(* CODESYS project IDE.xml
   cds-sync-save-after-import: True
   cds-sync-backup-name: cds-text-sync-reference-project
   cds-sync-enable-logging: True
   cds-text-sync-multipleApps: True
   cds-sync-backup-binary: True
   cds-sync-export-xml: True
   cds-sync-xml-first: True
   cds-sync-version: 1.7.5
   cds-sync-backup-retention-count: 3
   cds-sync-save-after-export: True
   cds-sync-safety-backup: True
   cds-sync-folder: C:\Workspace\Active\cds-text-sync-reference-project
   cds-sync-silent-mode: False
   cds-sync-pc: LOQ
   cds-daemon-config: {"poll_ms": 10, "deny": ["reset_plc", "reset_plc --kind origin", "create_boot_app", "plc_upload", "source_download"]}
   cds-sync-type-profile: codesys_sp20_plus

Project tree, tasks and I/O mapping:
  PLC : CODESYS Control Win V3 x64, CODESYS, version 3.5.20.10
    application ST_Application
      libraries: Standard, 3.5.22.0 (System); CAA CiA 405, 4.3.0.0 (CODESYS)
      task Task (cyclic, interval t#20ms, priority 1) calls ST_PROGRAMM, ST_PROGRAMM_AUX
      task Profinet_IOTask (cyclic, interval t#1ms, priority 1) calls nothing
      task Profinet_CommunicationTask (cyclic, interval t#10ms, priority 14) calls PN_Controller.CommCycle
      task EtherCAT_Task (cyclic, interval t#4ms, priority 1) calls nothing
      03_Object_POU_ST/
        01_PROGRAMM/
          program ST_PROGRAMM [ST]: ST_METHOD, ST_PROPERTY, ST_ACTION
          program ST_PROGRAMM_AUX [ST]
        02_FunctioanalBlock/
          function block ST_FB [ST]: ST_FB_Action, ST_FB_Method, ST_FB_Property
          function block ST_BLOCK_WITH_INTERFACE [ST]
        03_Function/
          function ST_Function [ST]
          function Empty_impementation_fn [ST]
          function fnBEETWEEN [ST]
        04_Interface/
          interface ITF_Base
          interface ITF_Child: Get_Value
      02_Object_GVL/
        declarations _02_TaskLocalGVL
        global variables _01_GVL
        global variables _03_NVL_sender
      01_Object_DUT/
        data type _04_DUT_UNION
        data type _02_DUT_Enumeration
        data type _03_DUT_Alias
        data type _01_DUT_STRUCTURE
        data type _01_DUT_STRUCTURE2
      04_additional/
        text list TextList
      Symbols
    application LD_Application
      libraries: Standard, 3.5.22.0 (System)
      task Task (cyclic, interval t#20ms, priority 1) calls LD_PROGRAMM, LD2_PROGRAMM
      03_Object_POU_LD/
        01_PROGRAMM/
          program LD_PROGRAMM [LD]
          program LD2_PROGRAMM [?]
        02_FunctionalBlock/
          function block LD_FB [LD]
        03_Function/
          function LD_Function [LD]
    application CFC_Application
      task Task (cyclic, interval t#20ms, priority 1) calls CFC_PROGRAMM, CFC_Page_PROGRAMM
      03_Object_POU_CFC/
        01_PROGRAMM/
          program CFC_PROGRAMM [CFC]
          program CFC_Page_PROGRAMM [CFC]
        02_FunctionalBlock/
          function block CFC_FB [CFC]
        03_Function/
          function CFC_R_TRIG [CFC]
      04_Persistent_vars/
      01_Object_DUT/
        data type _04_DUT_UNION
        data type _02_DUT_Enumeration
        data type _03_DUT_Alias
        data type _01_DUT_STRUCTURE
        data type _01_DUT_STRUCTURE2
    application FBD_Application
      libraries: Standard, 3.5.22.0 (System)
      task Task (cyclic, interval t#20ms, priority 1) calls nothing
      03_Object_POU_FBD/
        01_PROGRAMM/
        02_FunctionalBlock/
          function block FBD_FunctionBlock [FBD]: ST_Method_under_XML
        03_Function/
    Ethernet_Modbus : Ethernet, CODESYS, version 4.2.0.0
      Modbus_TCP_Client : Modbus TCP Client, CODESYS, version 4.5.0.0
        Modbus_TCP_Server : Modbus TCP Server, CODESYS, version 4.5.0.0
            settings: Unit-ID = 255; Channel 0.Function Code = 3; Channel 0.Read Offset = 16#0000; Channel 0.Read Length = 10; Channel 0.Write Offset = 0; Channel 0.Write Length = 0; Channel 0.Cycle Time = 100; Channel 1.Function Code = 16; Channel 1.Read Offset = 0; Channel 1.Read Length = 0; Channel 1.Write Offset = 16#0000; Channel 1.Write Length = 10; Channel 1.Cycle Time = 100
            unmapped channels: Channel 0, Channel 1
    Ethernet_Profinet : Ethernet, CODESYS, version 4.2.0.0
      PN_Controller : PN-Controller, CODESYS, order no. 1, version 4.7.1.0
          settings: First IP Address = [192, 168, 0, 2]; Last IP Address = [192, 168, 0, 254]; Default Subnet Mask = [255, 255, 255, 0]; Default Gateway Address = [0, 0, 0, 0]
        EL6631_0010_V2_0 : EL6631-0010 V2.0, Beckhoff, order no. EL6631-0010, version SW=V1.00, HW=V1.00
            settings: Slave parameters.Identification.IP address = [192,168,0,2]; Slave parameters.Identification.Subnet mask = [255,255,255,0]; Slave parameters.Identification.Default gateway = [0,0,0,0]; Slave parameters.Identification.MAC address = [16#00,16#00,16#00,16#00,16#00,16#00]; Slave parameters.Reduction ratio = 4; Slave parameters.Watchdog interval = 3
            unmapped channels: Inputs PS
    EtherCAT_Master : EtherCAT Master, CODESYS, version 4.10.0.0
      Unidrive_SP_Closed_Loop : Unidrive SP Closed Loop SoftMotion, Control Techniques, version 4.19.0.0
          settings: DC sync0 cycletime = 4000
          unmapped channels: Target Position, Control word, Modes of operation, Actual position, Status word, Modes of operation display
        SM_Drive_EtherCAT_ControlTechniques : SM_Drive_EtherCAT_ControlTechniques, CODESYS, order no. 0, version 4.19.0.0
            settings: wDriveID = 0; fSWMaxVelocity = 60; AddressOffset_8010 = 24; BitOffset_8010 = 0; BitLength_8010 = 16; Address_8010 = '%QW12'; Type_8010 = 'UINT'; AddressPointer_8010 = ADR(%QW12); AddressOffset_8020 = 26; BitOffset_8020 = 0; BitLength_8020 = 8; Address_8020 = '%QB26'; Type_8020 = 'USINT'; AddressPointer_8020 = ADR(%QB26); AddressOffset_8030 = 20; BitOffset_8030 = 0; BitLength_8030 = 32; Address_8030 = '%QD5'; Type_8030 = 'DINT'; AddressPointer_8030 = ADR(%QD5); AddressOffset_8510 = 28; BitOffset_8510 = 0; BitLength_8510 = 16; Address_8510 = '%IW14'; Type_8510 = 'UINT'; AddressPointer_8510 = ADR(%IW14); AddressOffset_8520 = 30; BitOffset_8520 = 0; BitLength_8520 = 8; Address_8520 = '%IB30'; Type_8520 = 'USINT'; AddressPointer_8520 = ADR(%IB30); AddressOffset_8530 = 24; BitOffset_8530 = 0; BitLength_8530 = 32; Address_8530 = '%ID6'; Type_8530 = 'DINT'; AddressPointer_8530 = ADR(%ID6)
    Modbus_COM_1 : Modbus COM, CODESYS, version 4.4.0.0
    Modbus_COM : Modbus COM, CODESYS, version 4.4.0.0
      Modbus_Client_COM_Port : Modbus Client, COM Port, CODESYS, version 4.5.0.0
        Modbus_Server_COM_Port : Modbus Server, COM Port, CODESYS, version 4.5.0.0
    CANbus : CANbus, CODESYS, version 4.3.0.0
      CANopen_Manager_SoftMotion : CANopen_Manager_SoftMotion, CODESYS, version 4.3.0.0
          settings: ConfigVersion = 50659584
        EPOS4_50_5 : EPOS4 50/5, maxon motor ag, order no. 000000, version 4.20.0.0
            settings: NODEIDSAVED = 1; SDO Timeout = 1000000; EXPERTSETTINGS = FALSE; Process by CANopenManager = TRUE; Process by CANopenManager = TRUE; PDO 16#1402.COBID = 16#00000401; PDO 16#1402.Transmission Type = 16#01; Process by CANopenManager = TRUE; Process by CANopenManager = TRUE; PDO 16#1800.COBID = 16#C0000181; PDO 16#1800.Event Timer = 0; Generic COBID = '$NODEID+16#C0000180'; Process by CANopenManager = TRUE; PDO 16#1801.COBID = 16#C0000281; PDO 16#1801.Event Timer = 0; Generic COBID = '$NODEID+16#C0000280'; Process by CANopenManager = TRUE; PDO 16#1802.Transmission Type = 16#01; PDO 16#1802.Event Timer = 0; Process by CANopenManager = TRUE; PDO 16#1803.COBID = 16#C0000481; PDO 16#1803.Event Timer = 0; Generic COBID = '$NODEID+16#C0000480'; Process by CANopenManager = TRUE; Controlword.Subindex = 16#00; Controlword.Subindex = 16#00; Modes of operation.Subindex = 16#00; Controlword.Subindex = 16#00; Target position.Subindex = 16#00; Controlword.Subindex = 16#00; Target velocity.Subindex = 16#00; Statusword.Subindex = 16#00; Statusword.Subindex = 16#00; Modes of operation display.Subindex = 16#00; Statusword.Subindex = 16#00; Position actual value.Subindex = 16#00; Statusword.Subindex = 16#00; Velocity actual value.Subindex = 16#00; SDO List.Set Heartbeat Consumer.Index = 16#1016; SDO List.Set Heartbeat Consumer.Subindex = 16#01;
              SDO List.Set Heartbeat Consumer.Value = 0; SDO List.Set Heartbeat Consumer.Size = 32; SDO List.Set Heartbeat Consumer.AbortIfError = FALSE; SDO List.Set Heartbeat Consumer.JumpToLine = FALSE; SDO List.Set Heartbeat Consumer.Line = 0; SDO List.Set Heartbeat Consumer.Index = 16#1016; SDO List.Set Heartbeat Consumer.Subindex = 16#02; SDO List.Set Heartbeat Consumer.Value = 0; SDO List.Set Heartbeat Consumer.Size = 32; SDO List.Set Heartbeat Consumer.AbortIfError = FALSE; SDO List.Set Heartbeat Consumer.JumpToLine = FALSE; SDO List.Set Heartbeat Consumer.Line = 0; SDO List.Set Heartbeat Producer.Index = 16#1017; SDO List.Set Heartbeat Producer.Subindex = 16#00; SDO List.Set Heartbeat Producer.Value = 16#00000000; SDO List.Set Heartbeat Producer.Size = 16; SDO List.Set Heartbeat Producer.AbortIfError = FALSE; SDO List.Set Heartbeat Producer.JumpToLine = FALSE; SDO List.Set Heartbeat Producer.Line = 0; SDO List.Disable PDO.Index = 16#1400; SDO List.Disable PDO.Subindex = 16#01; SDO List.Disable PDO.Value = 16#80000201; SDO List.Disable PDO.Size = 32; SDO List.Disable PDO.AbortIfError = FALSE; SDO List.Disable PDO.JumpToLine = FALSE; SDO List.Disable PDO.Line = 0; SDO List.Disable PDO.Index = 16#1401; SDO List.Disable PDO.Subindex = 16#01; SDO List.Disable PDO.Value = 16#80000301; SDO List.Disable PDO.Size = 32; SDO List.Disable PDO.AbortIfError = FALSE; SDO List.Disable PDO.JumpToLine = FALSE; SDO List.Disable PDO.Line = 0; SDO List.Disable PDO.Index = 16#1402; SDO List.Disable PDO.Subindex = 16#01; SDO List.Disable PDO.Value = 16#80000401; SDO List.Disable PDO.Size = 32; SDO List.Disable PDO.AbortIfError = FALSE; SDO List.Disable PDO.JumpToLine = FALSE; SDO List.Disable PDO.Line = 0;
              SDO List.Set transmission type.Index = 16#1402; SDO List.Set transmission type.Subindex = 16#02; SDO List.Set transmission type.Value = 16#01; SDO List.Set transmission type.Size = 8; SDO List.Set transmission type.AbortIfError = FALSE; SDO List.Set transmission type.JumpToLine = FALSE; SDO List.Set transmission type.Line = 0; SDO List.Clear pdo mapping.Index = 16#1602; SDO List.Clear pdo mapping.Subindex = 16#00; SDO List.Clear pdo mapping.Value = 16#0; SDO List.Clear pdo mapping.Size = 8; SDO List.Clear pdo mapping.AbortIfError = FALSE; SDO List.Clear pdo mapping.JumpToLine = FALSE; SDO List.Clear pdo mapping.Line = 0; SDO List.Set Mapping.Index = 16#1602; SDO List.Set Mapping.Subindex = 16#01; SDO List.Set Mapping.Value = 16#60400010; SDO List.Set Mapping.Size = 32; SDO List.Set Mapping.AbortIfError = FALSE; SDO List.Set Mapping.JumpToLine = FALSE; SDO List.Set Mapping.Line = 0; SDO List.Set Mapping.Index = 16#1602; SDO List.Set Mapping.Subindex = 16#02; SDO List.Set Mapping.Value = 16#607A0020; SDO List.Set Mapping.Size = 32; SDO List.Set Mapping.AbortIfError = FALSE; SDO List.Set Mapping.JumpToLine = FALSE; SDO List.Set Mapping.Line = 0; SDO List.Set number of mappings.Index = 16#1602; SDO List.Set number of mappings.Subindex = 16#00; SDO List.Set number of mappings.Value = 16#02; SDO List.Set number of mappings.Size = 8; SDO List.Set number of mappings.AbortIfError = FALSE; SDO List.Set number of mappings.JumpToLine = FALSE; SDO List.Set number of mappings.Line = 0; SDO List.Set and enable COB-ID.Index = 16#1402; SDO List.Set and enable COB-ID.Subindex = 16#01; SDO List.Set and enable COB-ID.Value = 16#00000401; SDO List.Set and enable COB-ID.Size = 32; SDO List.Set and enable COB-ID.AbortIfError = FALSE;
              SDO List.Set and enable COB-ID.JumpToLine = FALSE; SDO List.Set and enable COB-ID.Line = 0; SDO List.Disable PDO.Index = 16#1403; SDO List.Disable PDO.Subindex = 16#01; SDO List.Disable PDO.Value = 16#80000501; SDO List.Disable PDO.Size = 32; SDO List.Disable PDO.AbortIfError = FALSE; SDO List.Disable PDO.JumpToLine = FALSE; SDO List.Disable PDO.Line = 0; SDO List.Disable PDO.Index = 16#1800; SDO List.Disable PDO.Subindex = 16#01; SDO List.Disable PDO.Value = 16#C0000181; SDO List.Disable PDO.Size = 32; SDO List.Disable PDO.AbortIfError = FALSE; SDO List.Disable PDO.JumpToLine = FALSE; SDO List.Disable PDO.Line = 0; SDO List.Disable PDO.Index = 16#1801; SDO List.Disable PDO.Subindex = 16#01; SDO List.Disable PDO.Value = 16#C0000281; SDO List.Disable PDO.Size = 32; SDO List.Disable PDO.AbortIfError = FALSE; SDO List.Disable PDO.JumpToLine = FALSE; SDO List.Disable PDO.Line = 0; SDO List.Disable PDO.Index = 16#1802; SDO List.Disable PDO.Subindex = 16#01; SDO List.Disable PDO.Value = 16#C0000381; SDO List.Disable PDO.Size = 32; SDO List.Disable PDO.AbortIfError = FALSE; SDO List.Disable PDO.JumpToLine = FALSE; SDO List.Disable PDO.Line = 0; SDO List.Set transmission type.Index = 16#1802; SDO List.Set transmission type.Subindex = 16#02; SDO List.Set transmission type.Value = 16#01; SDO List.Set transmission type.Size = 8; SDO List.Set transmission type.AbortIfError = FALSE; SDO List.Set transmission type.JumpToLine = FALSE; SDO List.Set transmission type.Line = 0; SDO List.Set inhibit time.Index = 16#1802; SDO List.Set inhibit time.Subindex = 16#03; SDO List.Set inhibit time.Value = 16#000A;
              SDO List.Set inhibit time.Size = 16; SDO List.Set inhibit time.AbortIfError = FALSE; SDO List.Set inhibit time.JumpToLine = FALSE; SDO List.Set inhibit time.Line = 0; SDO List.Clear pdo mapping.Index = 16#1A02; SDO List.Clear pdo mapping.Subindex = 16#00; SDO List.Clear pdo mapping.Value = 16#0; SDO List.Clear pdo mapping.Size = 8; SDO List.Clear pdo mapping.AbortIfError = FALSE; SDO List.Clear pdo mapping.JumpToLine = FALSE; SDO List.Clear pdo mapping.Line = 0; SDO List.Set Mapping.Index = 16#1A02; SDO List.Set Mapping.Subindex = 16#01; SDO List.Set Mapping.Value = 16#60410010; SDO List.Set Mapping.Size = 32; SDO List.Set Mapping.AbortIfError = FALSE; SDO List.Set Mapping.JumpToLine = FALSE; SDO List.Set Mapping.Line = 0; SDO List.Set Mapping.Index = 16#1A02; SDO List.Set Mapping.Subindex = 16#02; SDO List.Set Mapping.Value = 16#60640020; SDO List.Set Mapping.Size = 32; SDO List.Set Mapping.AbortIfError = FALSE; SDO List.Set Mapping.JumpToLine = FALSE; SDO List.Set Mapping.Line = 0; SDO List.Set number of mappings.Index = 16#1A02; SDO List.Set number of mappings.Subindex = 16#00; SDO List.Set number of mappings.Value = 16#02; SDO List.Set number of mappings.Size = 8; SDO List.Set number of mappings.AbortIfError = FALSE; SDO List.Set number of mappings.JumpToLine = FALSE; SDO List.Set number of mappings.Line = 0; SDO List.Set and enable COB-ID.Index = 16#1802; SDO List.Set and enable COB-ID.Subindex = 16#01; SDO List.Set and enable COB-ID.Value = 16#40000381; SDO List.Set and enable COB-ID.Size = 32; SDO List.Set and enable COB-ID.AbortIfError = FALSE; SDO List.Set and enable COB-ID.JumpToLine = FALSE; SDO List.Set and enable COB-ID.Line = 0; SDO List.Disable PDO.Index = 16#1803;
              SDO List.Disable PDO.Subindex = 16#01; SDO List.Disable PDO.Value = 16#C0000481; SDO List.Disable PDO.Size = 32; SDO List.Disable PDO.AbortIfError = FALSE; SDO List.Disable PDO.JumpToLine = FALSE; SDO List.Disable PDO.Line = 0; ConfigVersion = 50659584
            unmapped channels: Controlword, Target position, Statusword, Position actual value
          SM3_Drive_CAN_Maxon_EPOS4 : SM3_Drive_CAN_Maxon_EPOS4, CODESYS, order no. 0, version 4.20.0.0
              settings: AdrOffset_8010 = 28; BitOffset_8010 = 0; BitLength_8010 = 16; Address_8010 = '%QW14'; Type_8010 = 'UINT'; AddressPointer_8010 = ADR(%QW14); AdrOffset_8020 = 32; BitOffset_8020 = 0; BitLength_8020 = 32; Address_8020 = '%QD8'; Type_8020 = 'DINT'; AddressPointer_8020 = ADR(%QD8); AdrOffset_8030 = 4294967295; BitOffset_8030 = 0; BitLength_8030 = 0; Address_8030 = ''; Type_8030 = ''; AddressPointer_8030 = 0; AdrOffset_8040 = 4294967295; BitOffset_8040 = 0; BitLength_8040 = 0; Address_8040 = ''; Type_8040 = ''; AddressPointer_8040 = 0; AdrOffset_8050 = 4294967295; BitOffset_8050 = 0; BitLength_8050 = 0; Address_8050 = ''; Type_8050 = ''; AddressPointer_8050 = 0; AdrOffset_8060 = 4294967295; BitOffset_8060 = 0; BitLength_8060 = 0; Address_8060 = ''; Type_8060 = ''; AddressPointer_8060 = 0; AdrOffset_8070 = 4294967295; BitOffset_8070 = 0; BitLength_8070 = 0; Address_8070 = '';
                Type_8070 = ''; AddressPointer_8070 = 0; AdrOffset_8080 = 4294967295; BitOffset_8080 = 0; BitLength_8080 = 0; Address_8080 = ''; Type_8080 = ''; AddressPointer_8080 = 0; AdrOffset_8090 = 4294967295; BitOffset_8090 = 0; BitLength_8090 = 0; Address_8090 = ''; Type_8090 = ''; AddressPointer_8090 = 0; AdrOffset_8510 = 32; BitOffset_8510 = 0; BitLength_8510 = 16; Address_8510 = '%IW16'; Type_8510 = 'UINT'; AddressPointer_8510 = ADR(%IW16); AdrOffset_8520 = 36; BitOffset_8520 = 0; BitLength_8520 = 32; Address_8520 = '%ID9'; Type_8520 = 'DINT'; AddressPointer_8520 = ADR(%ID9); AdrOffset_8530 = 4294967295; BitOffset_8530 = 0; BitLength_8530 = 0; Address_8530 = ''; Type_8530 = ''; AddressPointer_8530 = 0; AdrOffset_8540 = 4294967295; BitOffset_8540 = 0; BitLength_8540 = 0; Address_8540 = ''; Type_8540 = ''; AddressPointer_8540 = 0; AdrOffset_8550 = 4294967295; BitOffset_8550 = 0;
                BitLength_8550 = 0; Address_8550 = ''; Type_8550 = ''; AddressPointer_8550 = 0; AdrOffset_8560 = 4294967295; BitOffset_8560 = 0; BitLength_8560 = 0; Address_8560 = ''; Type_8560 = ''; AddressPointer_8560 = 0; AdrOffset_8570 = 4294967295; BitOffset_8570 = 0; BitLength_8570 = 0; Address_8570 = ''; Type_8570 = ''; AddressPointer_8570 = 0; AdrOffset_8580 = 4294967295; BitOffset_8580 = 0; BitLength_8580 = 0; Address_8580 = ''; Type_8580 = ''; AddressPointer_8580 = 0; AdrOffset_8590 = 4294967295; BitOffset_8590 = 0; BitLength_8590 = 0; Address_8590 = ''; Type_8590 = ''; AddressPointer_8590 = 0; AdrOffset_8600 = 4294967295; BitOffset_8600 = 0; BitLength_8600 = 0; Address_8600 = ''; Type_8600 = ''; AddressPointer_8600 = 0
            SM_Drive_Logical : SM_Drive_Logical, CODESYS, order no. 1805, version 4.14.0.0
                settings: wDriveID = 2
    SoftMotion General Axis Pool : SoftMotion General Axis Pool, CODESYS, version 4.11.0.0
  CODESYS_HMI : CODESYS HMI, CODESYS, order no. 311000, version 3.5.20.10
    application HMI_Application
      libraries: VisuDialogs, * (System)
      task VISU_TASK (cyclic, interval 200 ms, priority 31) calls VisuElems.Visu_Prg
      task Task (cyclic, interval t#20ms, priority 1) calls nothing
      task AlarmManagerTask (cyclic, interval 50 ms, priority 31) calls AlarmManager.Alarm_Prg
      Alarm Configuration
        alarm class Error (priority 10, acknowledge REP_ACK)
        alarm class Warning (priority 30, acknowledge REP)
        alarm class Info (priority 100, acknowledge REP)
        AlarmStorage
        alarm group AlarmGroup
            0 [Error]: Comparison Equal, ExpressionToCompare TRUE, Expression ZONE_HMI.arErrors[0] - "Error 1"
            1 [Warning]: Comparison Equal, ExpressionToCompare TRUE, Expression ZONE_HMI.arErrors[1] - "Warning 1"
        text list AlarmGroup
      MFL_VISU/
        global variables ZONE_HMI
        data type DUT_CONV_FRAME
        visualisation Screen
        visualisation FRAME_TWB
        data type ENUM_SegmentStatus
        visualisation Screen_1
      Symbols
  CODESYS_Linux_SL : CODESYS Control for Linux SL, CODESYS, order no. 2302000005, version 4.11.0.0
    application CI_CD_Application
      task Task (cyclic, interval t#4ms, priority 1) calls MAIN
      program MAIN [ST]
      FunctionBlocks/
        function block FB_Counter_UD [ST]
        function block FB_Delay [ST]
        function block FB_PulseTrain [ST]
        function block FB_TrafficLight [ST]
      Functions/
      GVL/
        global variables GVL_Test
      function block FB_Arithmetic [ST]
      function block FB_Checksum [ST]
      function block FB_Deadband [ST]
      function block FB_RangeCheck [ST]
      function block FB_Scale [ST]
    SoftMotion General Axis Pool
  text list GlobalTextList
*)

// PLC/ST_Application/01_Object_DUT/_04_DUT_UNION
TYPE _04_DUT_UNION :
UNION
	wValue : WORD;  // Overlaps iValue
	iValue : INT;   // Overlaps wValue
END_UNION
END_TYPE

// PLC/ST_Application/01_Object_DUT/_02_DUT_Enumeration
{attribute 'qualified_only'}
{attribute 'strict'}
TYPE _02_DUT_Enumeration :
(
	IDLE := 0,      // System waiting
	STARTING,       // Transition to running
	RUNNING,        // Active operation
	STOPPING,       // Controlled shutdown
	ERROR := 99     // Fault state
) INT;
END_TYPE

// PLC/ST_Application/01_Object_DUT/_03_DUT_Alias
TYPE _03_DUT_Alias : REAL; END_TYPE

// PLC/ST_Application/01_Object_DUT/_01_DUT_STRUCTURE
TYPE _01_DUT_STRUCTURE :
STRUCT
	sName : STRING(31);        // Pump designation
	rMaxFlow : REAL := 100.0;  // Capacity limit
	xIsVFD : BOOL;            // Has Variable Frequency Drive
	diWorkingHours : DINT;    // Total service time
END_STRUCT
END_TYPE

// PLC/ST_Application/01_Object_DUT/_01_DUT_STRUCTURE2
TYPE _01_DUT_STRUCTURE2 :
STRUCT
	sName : STRING(31);        // Pump designation
	rMaxFlow : REAL := 100.0;  // Capacity limit
	xIsVFD : BOOL;            // Has Variable Frequency Drive
	diWorkingHours : DINT;    // Total service time
END_STRUCT
END_TYPE

// PLC/CFC_Application/01_Object_DUT/_04_DUT_UNION
TYPE _04_DUT_UNION :
UNION
	wValue : WORD;  // Overlaps iValue
	iValue : INT;   // Overlaps wValue
END_UNION
END_TYPE

// PLC/CFC_Application/01_Object_DUT/_02_DUT_Enumeration
{attribute 'qualified_only'}
{attribute 'strict'}
TYPE _02_DUT_Enumeration :
(
	IDLE := 0,      // System waiting
	STARTING,       // Transition to running
	RUNNING,        // Active operation
	STOPPING,       // Controlled shutdown
	ERROR := 99     // Fault state
) INT;
END_TYPE

// PLC/CFC_Application/01_Object_DUT/_03_DUT_Alias
TYPE _03_DUT_Alias : REAL; END_TYPE

// PLC/CFC_Application/01_Object_DUT/_01_DUT_STRUCTURE
TYPE _01_DUT_STRUCTURE :
STRUCT
	sName : STRING(31);        // Pump designation
	rMaxFlow : REAL := 100.0;  // Capacity limit
	xIsVFD : BOOL;            // Has Variable Frequency Drive
	diWorkingHours : DINT;    // Total service time
END_STRUCT
END_TYPE

// PLC/CFC_Application/01_Object_DUT/_01_DUT_STRUCTURE2
TYPE _01_DUT_STRUCTURE2 :
STRUCT
	sName : STRING(31);        // Pump designation
	rMaxFlow : REAL := 100.0;  // Capacity limit
	xIsVFD : BOOL;            // Has Variable Frequency Drive
	diWorkingHours : DINT;    // Total service time
END_STRUCT
END_TYPE

// CODESYS_HMI/HMI_Application/MFL_VISU/DUT_CONV_FRAME
TYPE DUT_CONV_FRAME :
STRUCT
	conv_idx : INT := 1;      // Index in ZONE_MFL.g_aConfigs (1..4)
	sName : STRING(16);       // Safe name copy
	state : STRING(15);       // String representation of state
	//config : DUT_MFL_Config;  // Config copy for visualization
	dimension : INT := 50;    // [mm] segment size for ASCII
	pec_idx : USINT := 1;     // Which PEC to show slip for (1..10)
	iInstantSlip : INT;       // Current/Last measured slip [mm]
	
	// Compatibility fields for older Visu
	conv_number : INT; 
	pec_choice : INT;
	pecAverageSlip : INT;

	asciiString : STRING(255); // The visual representation
END_STRUCT
END_TYPE

// CODESYS_HMI/HMI_Application/MFL_VISU/ENUM_SegmentStatus
{attribute 'qualified_only'}
{attribute 'strict'}
TYPE ENUM_SegmentStatus :
(
	Empty_Segment := 95,     // '_' Empty 50mm space
	Cargo_Start := 91,       // '[' Left boundary of cargo item
	Cargo_End := 93,         // ']' Right boundary of cargo item
	Cargo_Filled := 35,      // '#' Segment fully occupied by cargo
	Sensor_Inactive := 111,  // 'o' Sensor position, no cargo detected
	Sensor_Active := 120,    // 'x' Sensor position, cargo detected
	Conveyor_Start := 123,   // '{'  Start edge of conveyor
	Conveyor_End := 125,     // '}' end edge of conveyor
	NULL := 0				 // String termination
)USINT;
END_TYPE

// PLC/ST_Application/02_Object_GVL/_02_TaskLocalGVL
// [INFO] Task with write access: Task (set manually in CODESYS, not restored by import)
{attribute 'qualified_only'}
VAR_GLOBAL
	iInteger : INT; // [INFO] Integer variable
END_VAR

// PLC/ST_Application/02_Object_GVL/_01_GVL
{attribute 'qualified_only'}
VAR_GLOBAL
END_VAR
VAR_GLOBAL
	xSysRestart : BOOL;         // Global system restart command
	rMainPressure : _03_DUT_Alias; // Using Alias type (renamed to match object)
	stActivePump : _01_DUT_STRUCTURE; // Using Structure type (renamed to match object)
	eCurrentState : _02_DUT_Enumeration; // Using Enum type (renamed to match object)
	uStatus : _04_DUT_UNION; // Using Union type (renamed to match object)
END_VAR

VAR_GLOBAL CONSTANT
	MAX_PUMPS : INT := 4;
	PI : REAL := 3.141592;
END_VAR

VAR_GLOBAL RETAIN
	diTotalCycleCounter : DINT; // Non-volatile counter
END_VAR

// PLC/ST_Application/02_Object_GVL/_03_NVL_sender
{attribute 'qualified_only'}
VAR_GLOBAL
	someInteger : INT; //Integer value
END_VAR

// CODESYS_HMI/HMI_Application/MFL_VISU/ZONE_HMI
{attribute 'qualified_only'}
VAR_GLOBAL
    // === Global Commands (HMI -> PLC) ===
    xStart: BOOL; // Master Start pulse for all zones
    xStop: BOOL; // Master Stop pulse for all zones
    xReset: BOOL; // Master Reset for all errors
    xReverse: BOOL; // Global direction control (Logic Level)
    xEmitt1: BOOL;
    xEmitt2: BOOL;


    // === Global Status (PLC -> HMI) ===
    xAnyError: BOOL; // True if any zone in error state
    xAnyWarning: BOOL; // True if any zone has a warning
    xSystemOK: BOOL; // True if communication and all zones are OK
    xRunning: BOOL; // True if at least one conveyor is moving

    // === Visualization Mapping ===
    // This array holds references to the frames used by the HMI.
    // It is initialized in MAIN.st to point to VISUALIZATION.aFrames.
    arConveyors: ARRAY[1..4] OF DUT_CONV_FRAME;
	
	arErrors : ARRAY[0..10] OF BOOL;

END_VAR

// CODESYS_Linux_SL/CI_CD_Application/GVL/GVL_Test
VAR_GLOBAL
	// Test flags for CI/CD
	g_xTestSuiteRunning : BOOL := FALSE;
	g_xAllPassed : BOOL := FALSE;
	g_uiTestCount : UINT := 0;
	g_uiPassCount : UINT := 0;
	g_uiFailCount : UINT := 0;
END_VAR

// PLC/ST_Application/03_Object_POU_ST/01_PROGRAMM/ST_PROGRAMM
PROGRAM ST_PROGRAMM
VAR_INPUT
	xEnable : BOOL;          // System enable
	xAutoMode : BOOL;        // Control mode: Auto (True) / Manual (False)
	rLevelSetpoint : REAL;   // Filling level setpoint
	rActualLevel : REAL;     // Current level (from sensor)
END_VAR

VAR_OUTPUT
	xPumpActive : BOOL;      // Output: Pump is active
	xLowLevelAlarm : BOOL;   // Output: Low level alarm
	rFlowRate : REAL;        // Current flow rate
END_VAR

VAR
	fbStartupDelay : TON;    // Startup delay timer
	xInternalError : BOOL;   // Internal error flag
	iStep : INT;             // Current algorithm step
	diGlobalStatus : DINT;   // System status (Moved from VAR_IN_OUT as PROGRAM doesn't support them when called by Task)
	iStartCounter : INT;     // Start counter (Moved from VAR_STAT as all variables in PROGRAM VAR are static by nature)
	iLevelStatus : INT;      // Level diagnostic status (from Method)
	xLevelOk : BOOL;         // Level validity flag (from Method)
	diOperatingHours : DINT; // Operating time in hours (via Property)
	xResetHours : BOOL;      // Manual command to reset hours (via Property)
	fbExample : ST_FB;       // Instance of the example Function Block
END_VAR

VAR_TEMP
	rLevelDiff : REAL;       // Temporary variable: level difference (reset every cycle)
END_VAR

VAR RETAIN
	diOperatingSeconds : DINT; // Retain variable: operating time (not reset on power loss)
END_VAR

VAR CONSTANT
	MAX_CAPACITY : REAL := 500.0; // Constant: maximum tank capacity
	MIN_LIMIT : REAL := 10.0;     // Constant: minimum limit threshold
END_VAR

// 0. Use Method to check if level is within safe range (0 to MAX_CAPACITY)
xLevelOk := ST_METHOD(rValue := rActualLevel,
                      rMin := 0.0,
                      rMax := MAX_CAPACITY,
                      iStatusCode => iLevelStatus);

// 1. Calculate level difference in temporary variable.
rLevelDiff := rLevelSetpoint - rActualLevel;
//Modificataion
// 2. Control logic
IF xEnable AND NOT xInternalError THEN

	IF xAutoMode THEN
		// Start pump based on setpoint with hysteresis
		IF rActualLevel < rLevelSetpoint - 5.0 AND NOT xPumpActive THEN
			fbStartupDelay(IN := TRUE, PT := T#2S);
			IF fbStartupDelay.Q THEN
				xPumpActive := TRUE;
				iStartCounter := iStartCounter + 1; // Update counter
			END_IF
		ELSIF rActualLevel >= rLevelSetpoint THEN
			xPumpActive := FALSE;
			fbStartupDelay(IN := FALSE);
		END_IF
	ELSE
		// In manual mode just monitor limits
		xPumpActive := xEnable AND (rActualLevel < MAX_CAPACITY);
	END_IF

ELSE
	xPumpActive := FALSE;
	fbStartupDelay(IN := FALSE);
END_IF

// 3. Alarm handling
xLowLevelAlarm := (rActualLevel < MIN_LIMIT);

// 4. Operating time accumulation (RETAIN)
IF xPumpActive THEN
	diOperatingSeconds := diOperatingSeconds + 1;
END_IF

// 5. Call Action to calculate flow
ST_ACTION();

// 6. Use Property to work with operating hours
diOperatingHours := ST_PROPERTY; // GET: Read hours converted from seconds

IF xResetHours THEN
    ST_PROPERTY := 0;            // SET: Reset seconds by setting property hours to 0
    xResetHours := FALSE;
END_IF

// 7. Status update
IF xLowLevelAlarm THEN
	diGlobalStatus := 999; // Error code
ELSIF xPumpActive THEN
	diGlobalStatus := 100; // Running
ELSE
	diGlobalStatus := 0;   // Standby
END_IF

// 8. Call example Function Block instance
fbExample(xEnable:= TRUE);
fbExample.ST_FB_Action();
fbExample.ST_FB_Method(iValueToAdd:= 1);

ST_Function(rValue:= 10.0, rMin:= 4.0, rMax:= 20.0);

METHOD ST_METHOD : BOOL
VAR_INPUT
	rValue : REAL;       // Value to check
	rMin : REAL;         // Minimum limit
	rMax : REAL;         // Maximum limit
END_VAR
VAR_OUTPUT
	iStatusCode : INT;   // 0: OK, 1: Too Low, 2: Too High
END_VAR
// This method checks if a value is within specified bounds

IF rValue < rMin THEN
	iStatusCode := 1;
	ST_METHOD := FALSE;
ELSIF rValue > rMax THEN
	iStatusCode := 2;
	ST_METHOD := FALSE;
ELSE
	iStatusCode := 0;
	ST_METHOD := TRUE;
END_IF
END_METHOD

PROPERTY ST_PROPERTY : DINT
GET
// Returns operating time in hours
ST_PROPERTY := diOperatingSeconds / 3600;
END_GET
SET
// Allows manual override/reset of operating seconds via hours
diOperatingSeconds := ST_PROPERTY * 3600;
END_SET
END_PROPERTY

ACTION ST_ACTION:
// This action simulates flow rate calculation based on pump activity
// Ideally called every cycle when pump is active

IF xPumpActive THEN
    // Simple simulation: flow increases until it reaches a nominal value
    IF rFlowRate < 45.5 THEN
        rFlowRate := rFlowRate + 0.5;
    ELSE
        rFlowRate := 45.5; // Nominal flow
    END_IF
ELSE
    // Flow drops when pump is off
    IF rFlowRate > 0.0 THEN
        rFlowRate := rFlowRate - 1.0;
    ELSE
        rFlowRate := 0.0;
    END_IF
END_IF
END_ACTION

END_PROGRAM

// PLC/ST_Application/03_Object_POU_ST/03_Function/ST_Function
FUNCTION ST_Function : BOOL
VAR_INPUT
	rValue : REAL;
	rMin : REAL;
	rMax : REAL;
END_VAR
VAR
END_VAR

IF rValue >= rMin AND rValue <= rMax THEN
	ST_Function := TRUE;
ELSE
	ST_Function := FALSE;//sd
END_IF

END_FUNCTION

// PLC/ST_Application/03_Object_POU_ST/02_FunctioanalBlock/ST_FB
FUNCTION_BLOCK ST_FB
VAR_INPUT
	xEnable : BOOL; // Enable counting
END_VAR
VAR_OUTPUT
	iCounter : INT; // Current counter value
	xLimitReached : BOOL; // Flag when limit is reached
END_VAR
VAR
	_iLimit : INT := 100; // Internal limit
END_VAR

IF xEnable THEN
	IF iCounter < _iLimit THEN
		iCounter := iCounter + 1;
		xLimitReached := FALSE;
	ELSE
		xLimitReached := TRUE;
	END_IF
ELSE
	xLimitReached := FALSE;
END_IF

ACTION ST_FB_Action:
iCounter := 0;
xLimitReached := FALSE;
END_ACTION

METHOD ST_FB_Method : BOOL
VAR_INPUT
	iValueToAdd : INT;
END_VAR
IF (iCounter + iValueToAdd) <= _iLimit THEN
	iCounter := iCounter + iValueToAdd;
	ST_FB_Method := TRUE;
ELSE
	ST_FB_Method := FALSE;
END_IF
END_METHOD

PROPERTY ST_FB_Property : INT
SET
_iLimit := ST_FB_Property;
END_SET
GET
ST_FB_Property := _iLimit;
END_GET
END_PROPERTY

END_FUNCTION_BLOCK

// PLC/ST_Application/03_Object_POU_ST/01_PROGRAMM/ST_PROGRAMM_AUX
PROGRAM ST_PROGRAMM_AUX
VAR
	diTotalHours : DINT;        // Total operating hours read from main program
	xMaintenanceReq : BOOL;    // Maintenance required flag
	iLogCounter : INT;         // Counter for log entries
	xBIT : BOOL;
END_VAR

VAR CONSTANT
	MAINTENANCE_INTERVAL : DINT := 1000; // Maintenance every 1000 hours
END_VAR

// 1. Accessing property of another program (ST_PROGRAMM)
// This is a GET access to the property in ST_PROGRAMM
diTotalHours := ST_PROGRAMM.ST_PROPERTY;

// 2. Logic to determine if maintenance is needed
IF diTotalHours >= MAINTENANCE_INTERVAL THEN
	xMaintenanceReq := TRUE;
ELSE
	xMaintenanceReq := FALSE;
END_IF

// 3. Example of direct variable access between programs.
// Reading a standard variable from ST_PROGRAMM
IF ST_PROGRAMM.xLowLevelAlarm AND iLogCounter < 100 THEN
    iLogCounter := iLogCounter + 1;
    // Here we could call a logging function
END_IF

// 4. Example of writing to another program
// We can reset the hours in the main program via its property
IF xMaintenanceReq AND ST_PROGRAMM.xAutoMode = FALSE THEN
    // Potentially reset hours after maintenance in manual mode
    // ST_PROGRAMM.ST_PROPERTY := 0; // SET access
END_IF

iLogCounter.0 := xBIT;

iLogCounter := BIT_TO_INT(xBIT);

END_PROGRAM

// CODESYS_Linux_SL/CI_CD_Application/MAIN
PROGRAM MAIN
VAR
	// CI/CD test instances â variables visible via read_variable/write_variable
	fbArith : FB_Arithmetic;
	fbScale : FB_Scale;
	fbDeadband : FB_Deadband;
	fbRangeCheck : FB_RangeCheck;
	fbChecksum : FB_Checksum;
	fbCounter : FB_Counter_UD;
END_VAR

// Pass-through call: inputs read from instance variables (set via online API),
// outputs written back to instance variables.
fbArith(rA := fbArith.rA, rB := fbArith.rB,
        eOp := fbArith.eOp, xExecute := fbArith.xExecute);

fbScale(rRaw := fbScale.rRaw, rRawMin := fbScale.rRawMin,
        rRawMax := fbScale.rRawMax, rScaledMin := fbScale.rScaledMin,
        rScaledMax := fbScale.rScaledMax, xExecute := fbScale.xExecute);

fbDeadband(rValue := fbDeadband.rValue, rBand := fbDeadband.rBand,
           xExecute := fbDeadband.xExecute);

fbRangeCheck(rValue := fbRangeCheck.rValue, rMin := fbRangeCheck.rMin,
             rMax := fbRangeCheck.rMax, xExecute := fbRangeCheck.xExecute);

fbChecksum(bA := fbChecksum.bA, bB := fbChecksum.bB,
           bC := fbChecksum.bC, xExecute := fbChecksum.xExecute);

fbCounter(xUp := fbCounter.xUp, xDown := fbCounter.xDown,
          xReset := fbCounter.xReset, uiLimit := fbCounter.uiLimit);

END_PROGRAM

// CODESYS_Linux_SL/CI_CD_Application/FB_Arithmetic
FUNCTION_BLOCK FB_Arithmetic
VAR_INPUT
	rA : REAL;
	rB : REAL;
	eOp : USINT; // 0=Add, 1=Sub, 2=Mul, 3=Div
	xExecute : BOOL;
END_VAR
VAR_OUTPUT
	rResult : REAL;
	xDone : BOOL;
END_VAR
VAR
	xPrev : BOOL;
END_VAR

IF xExecute AND NOT xPrev THEN
	CASE eOp OF
		0: rResult := rA + rB;
		1: rResult := rA - rB;
		2: rResult := rA * rB;
		3: 
			IF rB <> 0.0 THEN
				rResult := rA / rB;
			ELSE
				rResult := 0.0;
			END_IF
		ELSE
			rResult := 0.0;
	END_CASE
	xDone := TRUE;
END_IF

IF NOT xExecute THEN
	xDone := FALSE;
END_IF

xPrev := xExecute;

END_FUNCTION_BLOCK

// CODESYS_Linux_SL/CI_CD_Application/FB_Scale
FUNCTION_BLOCK FB_Scale
VAR_INPUT
	rRaw : REAL;
	rRawMin : REAL;
	rRawMax : REAL;
	rScaledMin : REAL;
	rScaledMax : REAL;
	xExecute : BOOL;
END_VAR
VAR_OUTPUT
	rResult : REAL;
	xDone : BOOL;
END_VAR
VAR
	xPrev : BOOL;
END_VAR

IF xExecute AND NOT xPrev THEN
	IF rRawMax <> rRawMin THEN
		rResult := rScaledMin + (rRaw - rRawMin) / (rRawMax - rRawMin) * (rScaledMax - rScaledMin);
	ELSE
		rResult := rScaledMin;
	END_IF
	// Clamp
	IF rResult < rScaledMin THEN rResult := rScaledMin; END_IF
	IF rResult > rScaledMax THEN rResult := rScaledMax; END_IF
	xDone := TRUE;
END_IF

IF NOT xExecute THEN
	xDone := FALSE;
END_IF

xPrev := xExecute;

END_FUNCTION_BLOCK

// CODESYS_Linux_SL/CI_CD_Application/FB_Deadband
FUNCTION_BLOCK FB_Deadband
VAR_INPUT
	rValue : REAL;
	rBand : REAL;
	xExecute : BOOL;
END_VAR
VAR_OUTPUT
	rResult : REAL;
	xDone : BOOL;
END_VAR
VAR
	xPrev : BOOL;
END_VAR

IF xExecute AND NOT xPrev THEN
	IF rValue >= -rBand AND rValue <= rBand THEN
		rResult := 0.0;
	ELSE
		rResult := rValue;
	END_IF
	xDone := TRUE;
END_IF

IF NOT xExecute THEN
	xDone := FALSE;
END_IF

xPrev := xExecute;

END_FUNCTION_BLOCK

// CODESYS_Linux_SL/CI_CD_Application/FB_RangeCheck
FUNCTION_BLOCK FB_RangeCheck
VAR_INPUT
	rValue : REAL;
	rMin : REAL;
	rMax : REAL;
	xExecute : BOOL;
END_VAR
VAR_OUTPUT
	xInRange : BOOL;
	xDone : BOOL;
END_VAR
VAR
	xPrev : BOOL;
END_VAR

IF xExecute AND NOT xPrev THEN
	xInRange := rValue >= rMin AND rValue <= rMax;
	xDone := TRUE;
END_IF

IF NOT xExecute THEN
	xDone := FALSE;
END_IF

xPrev := xExecute;

END_FUNCTION_BLOCK

// CODESYS_Linux_SL/CI_CD_Application/FB_Checksum
FUNCTION_BLOCK FB_Checksum
VAR_INPUT
	bA : BYTE;
	bB : BYTE;
	bC : BYTE;
	xExecute : BOOL;
END_VAR
VAR_OUTPUT
	bResult : BYTE;
	xDone : BOOL;
END_VAR
VAR
	xPrev : BOOL;
END_VAR

IF xExecute AND NOT xPrev THEN
	bResult := bA XOR bB XOR bC;
	xDone := TRUE;
END_IF

IF NOT xExecute THEN
	xDone := FALSE;
END_IF

xPrev := xExecute;

END_FUNCTION_BLOCK

// CODESYS_Linux_SL/CI_CD_Application/FunctionBlocks/FB_Counter_UD
FUNCTION_BLOCK FB_Counter_UD
VAR_INPUT
	xUp : BOOL := FALSE;
	xDown : BOOL := FALSE;
	xReset : BOOL := FALSE;
	uiLimit : UINT := 100;
END_VAR
VAR_OUTPUT
	uiValue : UINT := 0;
	xLimitReached : BOOL := FALSE;
END_VAR
VAR
	_xUpPrev : BOOL := FALSE;
	_xDownPrev : BOOL := FALSE;
END_VAR

// Reset
IF xReset THEN
	uiValue := 0;
	xLimitReached := FALSE;
	_xUpPrev := FALSE;
	_xDownPrev := FALSE;
	RETURN;
END_IF

// Rising edge up
IF xUp AND NOT _xUpPrev THEN
	IF uiValue < uiLimit THEN
		uiValue := uiValue + 1;
	END_IF
END_IF
_xUpPrev := xUp;

// Rising edge down
IF xDown AND NOT _xDownPrev THEN
	IF uiValue > 0 THEN
		uiValue := uiValue - 1;
	END_IF
END_IF
_xDownPrev := xDown;

// Limit detection
xLimitReached := uiValue >= uiLimit;

END_FUNCTION_BLOCK

// PLC/LD_Application/03_Object_POU_LD/01_PROGRAMM/LD_PROGRAMM
PROGRAM LD_PROGRAMM
VAR
	xStart : BOOL;
	xStop_NC : BOOL;
	xPump : BOOL;
	xLamp : BOOL;
	
	timer : TON;
	
	LD_FB_Instance : LD_FB;
END_VAR

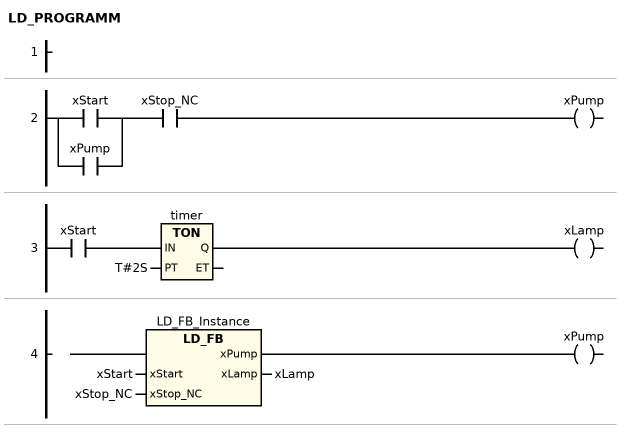
// NETWORK 1

// NETWORK 2
xPump := (xStart OR xPump) AND xStop_NC;

// NETWORK 3
timer(IN := xStart, PT := T#2S); // TON
xLamp := timer.Q;

// NETWORK 4
LD_FB_Instance(xStart := xStart, xStop_NC := xStop_NC, xLamp => xLamp); // LD_FB
xPump := LD_FB_Instance.xPump;

END_PROGRAM

// PLC/LD_Application/03_Object_POU_LD/02_FunctionalBlock/LD_FB
FUNCTION_BLOCK LD_FB
VAR_INPUT
	xStart : BOOL;
	xStop_NC : BOOL;
END_VAR
VAR_OUTPUT
	xPump : BOOL;
	xLamp : BOOL;
END_VAR
VAR
	
	
	
	timer : TON;
END_VAR

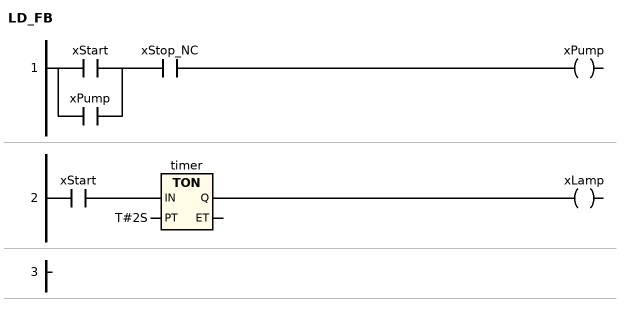
// NETWORK 1
xPump := (xStart OR xPump) AND xStop_NC;

// NETWORK 2
timer(IN := xStart, PT := T#2S); // TON
xLamp := timer.Q;

// NETWORK 3

END_FUNCTION_BLOCK

// PLC/LD_Application/03_Object_POU_LD/01_PROGRAMM/LD2_PROGRAMM
PROGRAM LD2_PROGRAMM
VAR
	xStart : BOOL;
	xStop_NC : BOOL;
	xPump : BOOL;
	xLamp : BOOL;
	
	timer : TON;
END_VAR

(* body of a kind this reader does not render *)

END_PROGRAM

// PLC/CFC_Application/03_Object_POU_CFC/01_PROGRAMM/CFC_PROGRAMM
PROGRAM CFC_PROGRAMM
VAR
	auxBool : BOOL;
	CLK : BOOL;
	R_TRIG_OUT : BOOL;
END_VAR
VAR_TEMP
	someBool : BOOL;
END_VAR
VAR // added by the converter: edge detectors and wires of the graphical bodies
    _w1, _w2 : ANY;
END_VAR

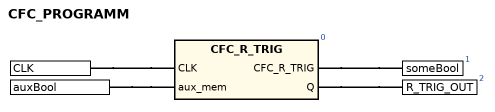
_w2 := CFC_R_TRIG(CLK := CLK, aux_mem := auxBool, Q => _w1);
someBool := _w2;
R_TRIG_OUT := _w1;

END_PROGRAM

// PLC/CFC_Application/03_Object_POU_CFC/03_Function/CFC_R_TRIG
FUNCTION CFC_R_TRIG : BOOL
VAR_INPUT
	CLK : BOOL;
END_VAR


VAR_IN_OUT
	aux_mem : BOOL;
END_VAR

VAR_OUTPUT
	Q : BOOL;
END_VAR

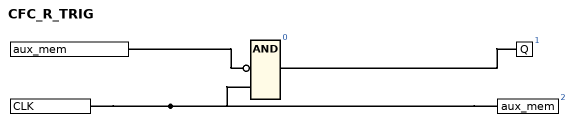
Q := NOT aux_mem AND CLK;
aux_mem := CLK;

END_FUNCTION

// PLC/CFC_Application/03_Object_POU_CFC/01_PROGRAMM/CFC_Page_PROGRAMM
PROGRAM CFC_Page_PROGRAMM
VAR
	auxBool : BOOL;
	CLK : BOOL;
	R_TRIG_OUT : BOOL;
END_VAR
VAR_TEMP
	someBool : BOOL;
END_VAR
VAR // added by the converter: edge detectors and wires of the graphical bodies
    _w1, _w2 : ANY;
END_VAR

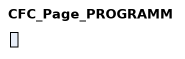
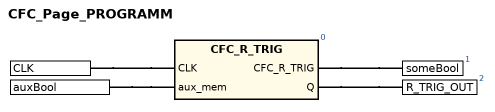
_w2 := CFC_R_TRIG(CLK := CLK, aux_mem := auxBool, Q => _w1);
someBool := _w2;
R_TRIG_OUT := _w1;

END_PROGRAM

// CODESYS_Linux_SL/CI_CD_Application/FunctionBlocks/FB_Delay
FUNCTION_BLOCK FB_Delay
VAR_INPUT
	xTrig : BOOL := FALSE;
	tDelay : TIME := T#1s;
END_VAR
VAR_OUTPUT
	xOut : BOOL := FALSE;
	xElapsed : BOOL := FALSE;
END_VAR
VAR
	_timer : TON;
	_xTrigPrev : BOOL := FALSE;
END_VAR

// Detect rising edge
IF xTrig AND NOT _xTrigPrev THEN
	_timer(IN := TRUE, PT := tDelay);
END_IF
_xTrigPrev := xTrig;

// Run timer
_timer();

xOut := _timer.Q;
xElapsed := _timer.Q AND NOT _xTrigPrev;

END_FUNCTION_BLOCK

// CODESYS_Linux_SL/CI_CD_Application/FunctionBlocks/FB_PulseTrain
FUNCTION_BLOCK FB_PulseTrain
VAR_INPUT
	xStart : BOOL := FALSE;
	xStop : BOOL := FALSE;
	uiPulseCount : UINT := 10;
	tPeriod : TIME := T#500ms;
END_VAR
VAR_OUTPUT
	xPulse : BOOL := FALSE;
	xBusy : BOOL := FALSE;
	xDone : BOOL := FALSE;
END_VAR
VAR
	_timer : TP;
	_pulseCount : UINT := 0;
	_xStartPrev : BOOL := FALSE;
	_running : BOOL := FALSE;
END_VAR

// Stop
IF xStop THEN
	_running := FALSE;
	_pulseCount := 0;
	xPulse := FALSE;
	xBusy := FALSE;
	xDone := FALSE;
	RETURN;
END_IF

// Start on rising edge
IF xStart AND NOT _xStartPrev THEN
	_running := TRUE;
	_pulseCount := 0;
	xDone := FALSE;
END_IF
_xStartPrev := xStart;

IF _running THEN
	_timer(IN := TRUE, PT := tPeriod);
	xPulse := _timer.Q;
	
	IF _timer.Q THEN
		_pulseCount := _pulseCount + 1;
		IF _pulseCount >= uiPulseCount THEN
			_running := FALSE;
			xDone := TRUE;
		END_IF
	END_IF
	
	xBusy := TRUE;
ELSE
	_timer(IN := FALSE);
	xPulse := FALSE;
	xBusy := FALSE;
END_IF

END_FUNCTION_BLOCK

// CODESYS_Linux_SL/CI_CD_Application/FunctionBlocks/FB_TrafficLight
FUNCTION_BLOCK FB_TrafficLight
VAR_INPUT
	xRun : BOOL := FALSE;
	xReset : BOOL := FALSE;
END_VAR
VAR_OUTPUT
	xRed : BOOL := FALSE;
	xYellow : BOOL := FALSE;
	xGreen : BOOL := FALSE;
	eState : USINT := 0; // 0=Red, 1=RedYellow, 2=Green, 3=Yellow
END_VAR
VAR
	_timer : TON;
	_state : USINT := 0;
	_times : ARRAY[0..3] OF TIME := [T#3s, T#1s, T#3s, T#1s];
	_xRunPrev : BOOL := FALSE;
END_VAR

IF xReset THEN
	_state := 0;
	xRed := FALSE; xYellow := FALSE; xGreen := FALSE;
	eState := 0;
	_timer(IN := FALSE);
	RETURN;
END_IF

// Start on rising edge
IF xRun AND NOT _xRunPrev THEN
	_state := 0;
	_timer(IN := TRUE, PT := _times[0]);
END_IF
_xRunPrev := xRun;

IF NOT xRun THEN
	_timer(IN := FALSE);
	xRed := FALSE; xYellow := FALSE; xGreen := FALSE;
	RETURN;
END_IF

// State machine
_timer();

IF _timer.Q THEN
	_state := (_state + 1) MOD 4;
	_timer(IN := TRUE, PT := _times[_state]);
END_IF

// Output mapping
CASE _state OF
	0: xRed := TRUE;  xYellow := FALSE; xGreen := FALSE;
	1: xRed := TRUE;  xYellow := TRUE;  xGreen := FALSE;
	2: xRed := FALSE; xYellow := FALSE; xGreen := TRUE;
	3: xRed := FALSE; xYellow := TRUE;  xGreen := FALSE;
END_CASE

eState := _state;

END_FUNCTION_BLOCK

// PLC/ST_Application/03_Object_POU_ST/02_FunctioanalBlock/ST_BLOCK_WITH_INTERFACE
FUNCTION_BLOCK ST_BLOCK_WITH_INTERFACE
VAR_INPUT
	someBOOL : BOOL; //commentary
END_VAR
VAR_OUTPUT
END_VAR
VAR
END_VAR

END_FUNCTION_BLOCK

// PLC/ST_Application/03_Object_POU_ST/03_Function/Empty_impementation_fn
FUNCTION Empty_impementation_fn : BOOL
VAR_INPUT
	SomeBool:BOOL;
END_VAR
VAR
END_VAR

END_FUNCTION

// PLC/ST_Application/03_Object_POU_ST/03_Function/fnBEETWEEN
FUNCTION fnBEETWEEN : BOOL
VAR_INPUT
	iValue : INT;
	iMin : INT;
	iMax : INT;
END_VAR
VAR
END_VAR

fnBEETWEEN := iValue >= iMin AND iValue <= iMax;

END_FUNCTION

// PLC/ST_Application/03_Object_POU_ST/04_Interface/ITF_Base
INTERFACE ITF_Base

END_INTERFACE

// PLC/ST_Application/03_Object_POU_ST/04_Interface/ITF_Child
INTERFACE ITF_Child EXTENDS ITF_Base

METHOD Get_Value
VAR_INPUT
END_VAR
END_METHOD

END_INTERFACE

// PLC/LD_Application/03_Object_POU_LD/03_Function/LD_Function
FUNCTION LD_Function : BOOL
VAR_INPUT
	xStart : BOOL;
	xStop_NC : BOOL;
END_VAR
VAR_OUTPUT
	xPump : BOOL;
END_VAR

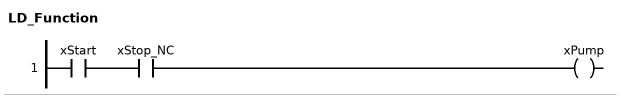
// NETWORK 1
xPump := xStart AND xStop_NC;

END_FUNCTION

// PLC/CFC_Application/03_Object_POU_CFC/02_FunctionalBlock/CFC_FB
FUNCTION_BLOCK CFC_FB
VAR_INPUT
END_VAR
VAR_OUTPUT
END_VAR
VAR
	auxBool : BOOL;
	CLK : BOOL;
	R_TRIG_OUT : BOOL;
END_VAR
VAR // added by the converter: edge detectors and wires of the graphical bodies
    _w1 : ANY;
END_VAR

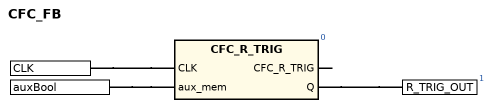
CFC_R_TRIG(CLK := CLK, aux_mem := auxBool, Q => _w1);
R_TRIG_OUT := _w1;

END_FUNCTION_BLOCK

// PLC/FBD_Application/03_Object_POU_FBD/02_FunctionalBlock/FBD_FunctionBlock
FUNCTION_BLOCK FBD_FunctionBlock
VAR_INPUT
	inINT : INT;
	bool1 : BOOL; //commented
	bool2 : BOOL;
END_VAR
VAR_OUTPUT
	outINT : INT;
	outBool : BOOL;
END_VAR
VAR
END_VAR

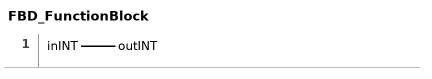
// NETWORK 1
outINT := inINT;

METHOD ST_Method_under_XML : BOOL
VAR_INPUT
END_VAR
ST_Method_under_XML := bool1 OR bool2;
//add comment123
END_METHOD

END_FUNCTION_BLOCK

// CODESYS_HMI/HMI_Application/MFL_VISU/Screen
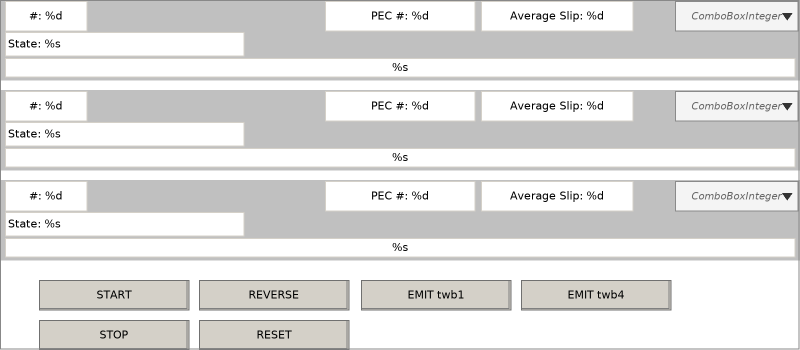
VISUALIZATION Screen  // 800x350
    Frame (0,0 800x80)
        shows FRAME_TWB(conveyor := ZONE_HMI.arConveyors[1])
    Frame (0,90 800x80)
        shows FRAME_TWB(conveyor := ZONE_HMI.arConveyors[2])
    Frame (0,180 800x80)
        shows FRAME_TWB(conveyor := ZONE_HMI.arConveyors[3])
    Button (39,280 150x30), "START"
        OnMouseClick: execute { ZONE_HMI.xStart := TRUE; }
    Button (199,280 150x30), "REVERSE"
        OnMouseClick:  ToggleVariable=ZONE_HMI.xReverse
    Button (361,280 150x30), "EMIT twb1"
        OnMouseClick:  ToggleVariable=ZONE_HMI.xEmitt1
    Button (521,280 150x30), "EMIT twb4"
        OnMouseClick:  ToggleVariable=ZONE_HMI.xEmitt2
    Button (39,320 150x30), "STOP"
        OnMouseClick: execute { ZONE_HMI.xStop := TRUE; }
    Button (199,320 150x30), "RESET"
        OnMouseClick: execute { ZONE_HMI.xReset := TRUE; }
END_VISUALIZATION

// CODESYS_HMI/HMI_Application/MFL_VISU/FRAME_TWB
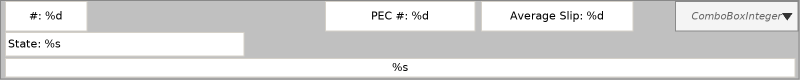
VISUALIZATION FRAME_TWB  // 800x80
VAR_IN_OUT
	conveyor : DUT_CONV_FRAME;
END_VAR
    Textfield (5,58 790x19), "%s", text variable: conveyor.asciiString
    ComboBoxInteger (675,1 123x30), variable: conveyor.dimension, text list: 'TextList_dimensions'
    Textfield (5,1 82x30), "#: %d", text variable: conveyor.conv_number
        OnMouseClick: write the text variable via Default, min 0, max 4
    Textfield (325,1 150x30), "PEC #: %d", text variable: conveyor.pec_idx
        OnMouseClick: write the text variable via Default, min 1, max 10
    Textfield (481,1 152x30), "Average Slip: %d", text variable: conveyor.pecAverageSlip
    Textfield (5,32 239x24), "State: %s", text variable: conveyor.state
END_VISUALIZATION

// CODESYS_HMI/HMI_Application/MFL_VISU/Screen_1
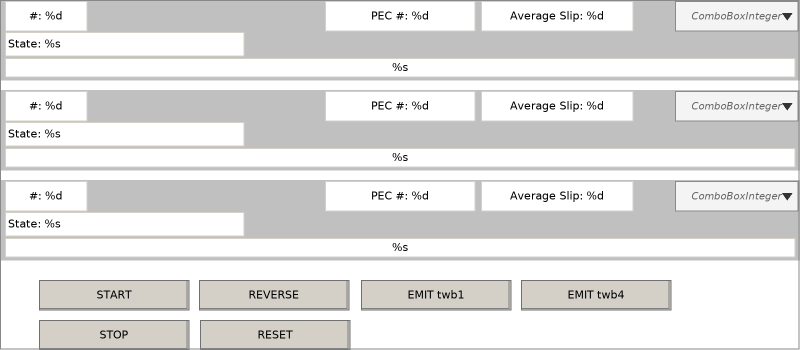
VISUALIZATION Screen_1  // 800x350
    Frame (0,0 800x80)
        shows FRAME_TWB(conveyor := ZONE_HMI.arConveyors[1])
    Frame (0,90 800x80)
        shows FRAME_TWB(conveyor := ZONE_HMI.arConveyors[2])
    Frame (0,180 800x80)
        shows FRAME_TWB(conveyor := ZONE_HMI.arConveyors[3])
    Button (39,280 150x30), "START"
        OnMouseClick: execute { ZONE_HMI.xStart := TRUE; }
    Button (199,280 150x30), "REVERSE"
        OnMouseClick:  ToggleVariable=ZONE_HMI.xReverse
    Button (361,280 150x30), "EMIT twb1"
        OnMouseClick:  ToggleVariable=ZONE_HMI.xEmitt1
    Button (521,280 150x30), "EMIT twb4"
        OnMouseClick:  ToggleVariable=ZONE_HMI.xEmitt2
    Button (39,320 150x30), "STOP"
        OnMouseClick: execute { ZONE_HMI.xStop := TRUE; }
    Button (200,320 150x30), "RESET"
        OnMouseClick: execute { ZONE_HMI.xReset := TRUE; }
END_VISUALIZATION

(* text list TextList (id | default)
  0 | Default
  1 | First
  2 | Second
  3 | Third
   |  *)

(* text list AlarmGroup (id | default)
  1 | Warning 1
  0 | Error 1
   |  *)
